ABB RAPID module: TCP_Sergiox2f.MOD

MODULE TCP_Sergiox2f
	! Points are read in order of declaration.
  ! Please do not change the order of points!

  LOCAL PERS robtarget pTCP_Point1:=[[447.3126,44.52092,202.975],[0.424976468086243,-0.277205526828766,0.844860255718231,-0.169597074389458],[0,0,-1,1],[9E+09,9E+09,9E+09,9E+09,9E+09,9E+09]];
	LOCAL PERS robtarget pTCP_Point2:=[[585.0396,192.0515,188.9114],[0.229034677147865,0.378602832555771,0.781667530536652,-0.439543932676315],[0,1,-1,1],[9E+09,9E+09,9E+09,9E+09,9E+09,9E+09]];
	LOCAL PERS robtarget pTCP_Point3:=[[720.9886,74.21651,224.5959],[0.0140435406938195,0.886993885040283,0.265147119760513,-0.377811640501022],[0,1,-1,1],[9E+09,9E+09,9E+09,9E+09,9E+09,9E+09]];
	LOCAL PERS robtarget pTCP_Point4:=[[591.9858,-102.7634,202.1752],[0.411151111125946,-0.795599639415741,0.401147693395615,0.192500308156013],[-1,-2,0,1],[9E+09,9E+09,9E+09,9E+09,9E+09,9E+09]];

ENDMODULE
